PROGRAM MAIN
VAR
	_sampleContext 				: 	TcoCognexVision.SampleContext;
	_sampleComponentTests 		:	SampleComponentTests;
	_tcoDataman_v_5_x_xTests 	:	TcoDataman_v_5_x_xTests;
END_VAR

_sampleContext.Run();
_sampleComponentTests.Run();
_tcoDataman_v_5_x_xTests.Run();

END_PROGRAM

(* stored: Version 1.1.0.1, ProductVersion 3.1.4024.11
   POU MAIN: Id {5b53fb17-cd82-0ea5-175c-64a7847dafcb}, SpecialFunc None *)
